FUNCTION F_Limit : BOOL
VAR_INPUT
    fVal : LREAL;
    fLLim : LREAL;
    fHLim : LREAL;
    bInclusive : BOOL;
END_VAR
VAR
END_VAR


IF bInclusive THEN
    IF fLLim <= fHLim THEN
        F_Limit := fLLim <= fVal AND fHLim >= fVal;
    ELSE
        F_Limit := fLLim >= fVal OR fHLim <= fVal;
    END_IF
ELSE
    IF fLLim <= fHLim THEN
        F_Limit := fLLim < fVal AND fHLim > fVal;
    ELSE
        F_Limit := fLLim > fVal OR fHLim < fVal;
    END_IF
END_IF

END_FUNCTION

(* stored: Version 1.1.0.1
   POU F_Limit: Id {110c4ed8-1696-490e-8f8e-19d67e06929f}, SpecialFunc None *)
